// TIA Portal V18 export
DATA_BLOCK "Display_management_DB"   // DB17
VERSION : 0.1
// stored: AutoNumber true, InstanceOfName Display_management, InstanceOfType FB
"Display_management"
   // VAR
   //    HMI_In_selection_handling_Instance { S7_SetPoint := 'True'} : "HMI_In_selection_handling";
   //    HMI_In_selection_handling_Instance_1 { S7_SetPoint := 'True'} : "HMI_In_selection_handling";
   //    HMI_In_selection_handling_Instance_2 { S7_SetPoint := 'True'} : "HMI_In_selection_handling";
   //    HMI_In_selection_handling_Instance_3 { S7_SetPoint := 'True'} : "HMI_In_selection_handling";
   //    HMI_In_selection_handling_Instance_4 { S7_SetPoint := 'True'} : "HMI_In_selection_handling";
   //    HMI_In_selection_handling_Instance_5 { S7_SetPoint := 'True'} : "HMI_In_selection_handling";
   //    HMI_In_selection_handling_Instance_6 { S7_SetPoint := 'True'} : "HMI_In_selection_handling";
   //    HMI_In_selection_handling_Instance_7 { S7_SetPoint := 'True'} : "HMI_In_selection_handling";
   // END_VAR
BEGIN
END_DATA_BLOCK
